{attribute 'GeneratedUsingTerminal: EK1122-0000-0018'}
{attribute addProperty BoxType "EK1122-0000-0018"}
{attribute addProperty Id "Beckhoff_EL9xxxsub_EK1100EK1100_1FC0878B2"}
{attribute addProperty CRC "220869795"}
{attribute addProperty Size "2"}
TYPE Beckhoff_EL9xxxEK1122_0D2A34A3 EXTENDS EK1122_1FC0878B :
STRUCT
	{attribute addProperty Name "Beckhoff_EL9xxxsub_EK1100"}
	{attribute addProperty PreviousPort "Beckhoff EL9xxxEK1122 : D"}
	Beckhoff_EL9xxxsub_EK1100 : EK1100_1FC0878B;
END_STRUCT
END_TYPE

(* stored: Version 1.2.0.0, ProductVersion 3.1.4024.9
   DUT Beckhoff_EL9xxxEK1122_0D2A34A3: Id {d747db52-acc0-4111-aff8-b605d1147d91} *)
